TYPE ST_Event :
STRUCT
	eEventType : E_TcEventClass;
	eEventSeverity : TcEventSeverity;
	nEventID : UDINT;
	sEventDescription : STRING(255);
	dtTimestamp : DATE_AND_TIME;
END_STRUCT
END_TYPE

(* stored: Version 1.1.0.1, ProductVersion 3.1.4024.10
   DUT ST_Event: Id {0600e0e7-89f9-41fc-9b2d-7f9e558decf6} *)
